FUNCTION_BLOCK FB_hmi_connection
VAR_INPUT
	//Initlize datagrid params
	payoff_input_datagrid_params_list: ARRAY[1..GVL.MAX_PAYOFF_COUNT] OF payoff_input_datagrid_params;
	payoff_output_datagrid_params_list: ARRAY[1..GVL.MAX_PAYOFF_COUNT] OF payoff_output_datagrid_params;
	pickup_input_datagrid_params_list: ARRAY[1..GVL.MAX_PICKUP_COUNT] OF pickup_input_datagrid_params;
	pickup_output_datagrid_params_list: ARRAY[1..GVL.MAX_PICKUP_COUNT] OF pickup_output_datagrid_params;
	general_input_datagrid_params_list: ARRAY[1..1] OF general_input_datagrid_params;
	misc_settings_input_datagrid_params_list :ARRAY[1..1] OF misc_settings_input_datagrid_params;
	pickup_pancake_input_datagrid_params_list : ARRAY[1..1] OF pancake_params_0;
	pickup_racetrack_input_datagrid_params_list : ARRAY[1..1] OF racetrack_params_1;
	output_error_datagrid_list : ARRAY[0..3] OF output_error_datagrid;
	motor_state_datagrid_list : ARRAY[0..3] OF motor_state_datagrid;
	overview_outputs_datagrid_list :ARRAY[1..1] OF overview_outputs_datagrid;
	
	color_list :ARRAY[0..3] OF DWORD;
	//Outputs
	
	motor_turncount : ARRAY[1..4] of DINT;
	
	
	
	//HARDWARE INPUTS
	
	estopHW AT %I* : BOOL := FALSE;
	
	//CONTROL PAGE
	resetUI : BOOL ;
	startUI : BOOL ;
	tensionUI : BOOL;
	homeUI : BOOL;
	
	//SETTINGS
	checkInputsUI : BOOL;
	updateInputsUI : BOOL;
	
	//OUTPUT
	clearUI : BOOL;
	
	//HISTORYIZED VARS
	torque : ARRAY[1..GVL.MAX_PAYOFF_COUNT+GVL.MAX_PICKUP_COUNT] OF LREAL;
	rpm : ARRAY[1..GVL.MAX_PAYOFF_COUNT+GVL.MAX_PICKUP_COUNT] OF LREAL;
	
	//misc
	state : INT:=0;
	
END_VAR

METHOD CYCLIC : BOOL
VAR_INPUT
END_VAR

VAR

END_VAR
END_METHOD

METHOD INIT : BOOL
VAR_INPUT
END_VAR
init_datagrids();
END_METHOD

METHOD init_datagrids : BOOL
VAR_INPUT
END_VAR

VAR
	i: INT;
END_VAR
//initalize datagrids for ui
FOR i := 1 TO GVL.MAX_PAYOFF_COUNT DO
	
	payoff_input_datagrid_params_list[i].motor_name := TO_STRING(i);
	payoff_output_datagrid_params_list[i].motor_name := TO_STRING(i);
		
END_FOR;

pickup_input_datagrid_params_list[1].motor_name := TO_STRING(1);
pickup_output_datagrid_params_list[1].motor_name := TO_STRING(1);
END_METHOD

END_FUNCTION_BLOCK

(* stored: Version 1.1.0.1, ProductVersion 3.1.4024.12
   POU FB_hmi_connection: Id {16fd796a-42c3-43cf-88b6-53e67b78becc}, SpecialFunc None
   Folder Methods: Id {9718d345-c687-4cc8-aec1-c0b0c29132ec}
   Method CYCLIC: Id {e0324688-916e-4bfe-98af-5869031e350d}
   Method INIT: Id {380bcd9f-89dd-442f-8edd-b047340f0d4e}
   Method init_datagrids: Id {9e027757-0043-4a80-8af8-6e4796c997e6} *)
